Staubli VAL3: test_ventouse.pgx

program test_ventouse()
begin
  open(ventouse)
  movej(jP1, ventouse, mNomSpeed)
  movej(jP2, ventouse, mNomSpeed)
  close(ventouse)
  movej(jP4, ventouse, mNomSpeed)
  movej(jP5, ventouse, mNomSpeed)
  movej(jP3, ventouse, mNomSpeed)
  open(ventouse)
  movej(jP1, ventouse, mNomSpeed)
  movej(jP3, ventouse, mNomSpeed)
  close(ventouse)
  movej(jP5, ventouse, mNomSpeed)
  movej(jP4, ventouse, mNomSpeed)
  movej(jP2, ventouse, mNomSpeed)
  open(ventouse)
  waitEndMove()
end
